{attribute 'GeneratedUsingTerminal: EL2912-0000-0016'}
{attribute addProperty BoxType "EL2912-0000-0016"}
{attribute addProperty Id "FSoE_InputsFSoE_Inputs_939ABF3D7FSoE_OutputsFSoE_Outputs_3899B1859"}
{attribute addProperty CRC "641013422"}
{attribute addProperty Size "16"}
TYPE Module_1_FSOE_263516AE :
STRUCT
	{attribute addProperty Name "FSoE_Inputs"}
	FSoE_Inputs  : FSoE_Inputs_939ABF3D;
	{attribute addProperty Name "FSoE_Outputs"}
	FSoE_Outputs  : FSoE_Outputs_3899B185;
END_STRUCT
END_TYPE

(* stored: Version 1.2.0.0, ProductVersion 3.1.4024.9
   DUT Module_1_FSOE_263516AE: Id {5fcfb19b-e28b-46f5-ae7c-ec78e462a9a2} *)
